FUNCTION_BLOCK Station1Skill (* Basic FB with empty ECC *)
  (* Standard: 61499-2 *)
  (* Version 1.0, 2021-09-15, dorofeev *)
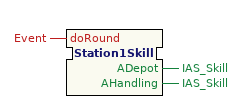
  EVENT_INPUT
    doRound;
  END_EVENT
  PLUGS
    ADepot : IAS_Skill;
    AHandling : IAS_Skill;
  END_PLUGS
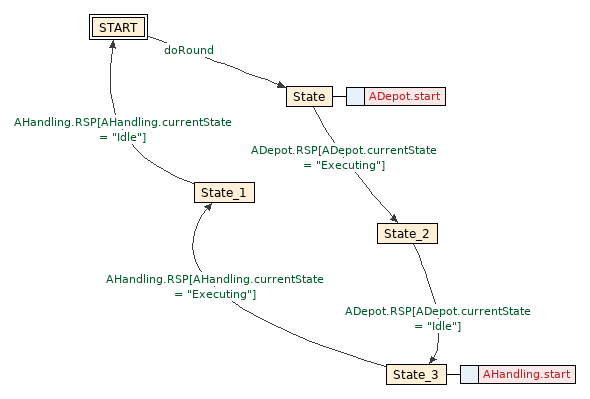
  EC_STATES
    START; (* Initial State *)
    State : -> ADepot.start;
    State_1;
    State_2;
    State_3 : -> AHandling.start;
  END_STATES
  EC_TRANSITIONS
    START TO State := doRound;
    State_1 TO START := AHandling.RSP[AHandling.currentState = "Idle"];
    State TO State_2 := ADepot.RSP[ADepot.currentState = "Executing"];
    State_2 TO State_3 := ADepot.RSP[ADepot.currentState = "Idle"];
    State_3 TO State_1 := AHandling.RSP[AHandling.currentState = "Executing"];
  END_TRANSITIONS
END_FUNCTION_BLOCK
